PROGRAM MAIN
VAR
	(*
	fbReadRegs        : FB_MBReadRegs;
    bReadRegs         : BOOL;
    bReadRegsBusy     : BOOL;
    bReadRegsError    : BOOL;
    nReadRegsErrorId  : UDINT;
    nReadRegsCount    : UDINT;
    nQuantity         : WORD:=2;
    nMBAddr           : WORD:=24;
    arrData           : ARRAY [1..2] OF WORD;
	*)
	
	//myBlink	: Array[0..7] OF MyBlink();
	redBlink	: MyBlink();
	yellowBlink	: MyBlink();
	greenBlink	: MyBlink();
	controlPanel 	:	ControlPanel();
	
END_VAR

Blink();


ControlPanel();

END_PROGRAM

(* stored: Version 1.1.0.1, ProductVersion 3.1.4024.12
   POU MAIN: Id {761fd973-c8da-4c7a-9c6a-57bff7cf3149}, SpecialFunc None *)
